{attribute 'GeneratedUsingTerminal: EL9187--0000'}
{attribute addProperty BoxType "EL9187--0000"}
{attribute addProperty Description "EL9187 Potential Connection, 8 x Ground"}
{attribute addProperty Physics "KK"}
{attribute addProperty Id "EL9187"}
{attribute addProperty CRC "2505203337"}
{attribute addProperty Size "0"}
TYPE EL9187_95525E89 EXTENDS EtcSlaveTerminalBase_947E5A46 :
STRUCT
END_STRUCT
END_TYPE

(* stored: Version 1.2.0.0, ProductVersion 3.1.4024.11
   DUT EL9187_95525E89: Id {b2fc2b4d-0959-4d77-99cb-7779363106a6} *)
